PROGRAM MAIN
VAR
	fbLightController	: FB_LightController;
END_VAR
VAR CONSTANT
	NUMBER_OF_REG_LIGHTS		: USINT := 4;
	NUMBER_OF_DIMMABLE_LIGHTS	: USINT := 4;
	MAXIMUM_NUMBER_OF_LIGHTS	: USINT := NUMBER_OF_DIMMABLE_LIGHTS + NUMBER_OF_REG_LIGHTS;
END_VAR

fbLightController();

END_PROGRAM

(* stored: Version 1.1.0.1, ProductVersion 3.1.4024.12
   POU MAIN: Id {dcb8f025-7b78-44de-a3ef-76b85cfb3e40}, SpecialFunc None *)
